FUNCTION_BLOCK alarmeHH_H_L_LL (* Composite Function Block Type *)
  (* Standard: 61499-2 *)
  (* Version 0.0, 1/23/2026, Schneider Electric, template *)
  PACKAGE Hidryco.HidrycoLib;
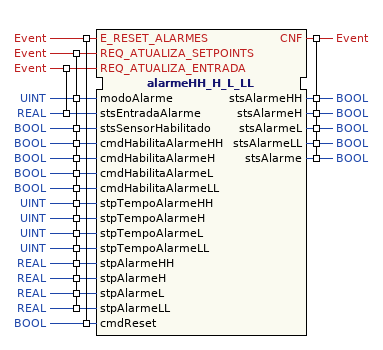
  EVENT_INPUT
    E_RESET_ALARMES WITH cmdReset;
    REQ_ATUALIZA_SETPOINTS WITH modoAlarme, cmdHabilitaAlarmeHH, cmdHabilitaAlarmeH, cmdHabilitaAlarmeL, cmdHabilitaAlarmeLL, stpTempoAlarmeHH, stpTempoAlarmeH, stpTempoAlarmeL, stpTempoAlarmeLL, stpAlarmeHH, stpAlarmeH, stpAlarmeL, stpAlarmeLL, stsSensorHabilitado;
    REQ_ATUALIZA_ENTRADA WITH stsEntradaAlarme;
  END_EVENT
  EVENT_OUTPUT
    CNF WITH stsAlarmeHH, stsAlarmeH, stsAlarmeL, stsAlarmeLL, stsAlarme; (* Execution Confirmation *)
  END_EVENT
  VAR_INPUT
    modoAlarme : UINT; (* 0 - AutoReset, 1 - Comando Reset *)
    stsEntradaAlarme : REAL;
    stsSensorHabilitado : BOOL;
    cmdHabilitaAlarmeHH : BOOL;
    cmdHabilitaAlarmeH : BOOL;
    cmdHabilitaAlarmeL : BOOL;
    cmdHabilitaAlarmeLL : BOOL;
    stpTempoAlarmeHH : UINT;
    stpTempoAlarmeH : UINT;
    stpTempoAlarmeL : UINT;
    stpTempoAlarmeLL : UINT;
    stpAlarmeHH : REAL;
    stpAlarmeH : REAL;
    stpAlarmeL : REAL;
    stpAlarmeLL : REAL;
    cmdReset : BOOL;
  END_VAR
  VAR_OUTPUT
    stsAlarmeHH : BOOL; (* Output event qualifier *)
    stsAlarmeH : BOOL;
    stsAlarmeL : BOOL;
    stsAlarmeLL : BOOL;
    stsAlarme : BOOL;
  END_VAR
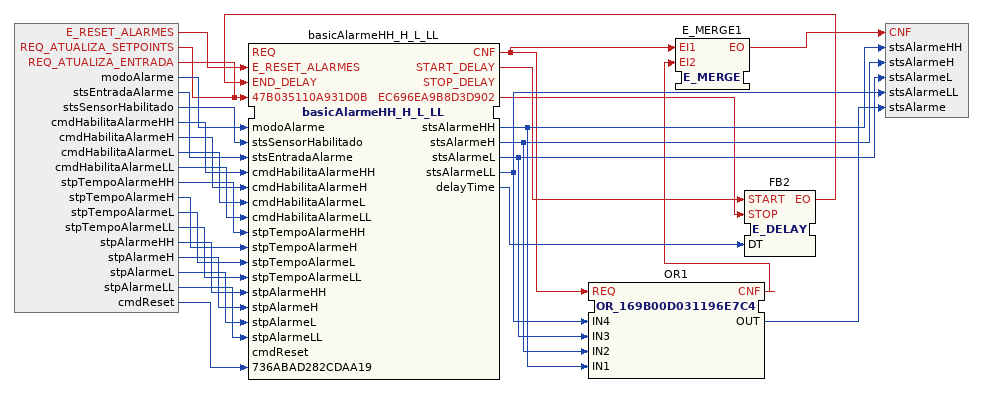
  FBS
    basicAlarmeHH_H_L_LL : basicAlarmeHH_H_L_LL;
    FB2 : E_DELAY;
    OR1 : OR_169B00D031196E7C4; {SET_ATTRIBUTE(Configuration.GenericFBType.InterfaceParams, Runtime.Standard#CNT:=4;OUT:BOOL)}
    E_MERGE1 : E_MERGE;
  END_FBS
  EVENT_CONNECTIONS
    basicAlarmeHH_H_L_LL.START_DELAY TO FB2.START;
    FB2.EO TO basicAlarmeHH_H_L_LL.END_DELAY;
    E_RESET_ALARMES TO basicAlarmeHH_H_L_LL.E_RESET_ALARMES;
    basicAlarmeHH_H_L_LL.CNF TO E_MERGE1.EI1;
    basicAlarmeHH_H_L_LL.CNF TO OR1.REQ;
    OR1.CNF TO E_MERGE1.EI2;
    E_MERGE1.EO TO CNF;
    REQ_ATUALIZA_SETPOINTS TO basicAlarmeHH_H_L_LL.47B035110A931D0B;
    REQ_ATUALIZA_ENTRADA TO basicAlarmeHH_H_L_LL.47B035110A931D0B;
    basicAlarmeHH_H_L_LL.EC696EA9B8D3D902 TO FB2.STOP;
  END_CONNECTIONS
  DATA_CONNECTIONS
    basicAlarmeHH_H_L_LL.delayTime TO FB2.DT;
    basicAlarmeHH_H_L_LL.stsAlarmeLL TO stsAlarmeLL;
    basicAlarmeHH_H_L_LL.stsAlarmeL TO stsAlarmeL;
    basicAlarmeHH_H_L_LL.stsAlarmeH TO stsAlarmeH;
    basicAlarmeHH_H_L_LL.stsAlarmeHH TO stsAlarmeHH;
    modoAlarme TO basicAlarmeHH_H_L_LL.modoAlarme;
    cmdHabilitaAlarmeHH TO basicAlarmeHH_H_L_LL.cmdHabilitaAlarmeHH;
    cmdHabilitaAlarmeH TO basicAlarmeHH_H_L_LL.cmdHabilitaAlarmeH;
    cmdHabilitaAlarmeL TO basicAlarmeHH_H_L_LL.cmdHabilitaAlarmeL;
    cmdHabilitaAlarmeLL TO basicAlarmeHH_H_L_LL.cmdHabilitaAlarmeLL;
    stpTempoAlarmeHH TO basicAlarmeHH_H_L_LL.stpTempoAlarmeHH;
    stpTempoAlarmeH TO basicAlarmeHH_H_L_LL.stpTempoAlarmeH;
    stpTempoAlarmeL TO basicAlarmeHH_H_L_LL.stpTempoAlarmeL;
    stpTempoAlarmeLL TO basicAlarmeHH_H_L_LL.stpTempoAlarmeLL;
    stpAlarmeHH TO basicAlarmeHH_H_L_LL.stpAlarmeHH;
    stpAlarmeH TO basicAlarmeHH_H_L_LL.stpAlarmeH;
    stpAlarmeL TO basicAlarmeHH_H_L_LL.stpAlarmeL;
    stpAlarmeLL TO basicAlarmeHH_H_L_LL.stpAlarmeLL;
    stsEntradaAlarme TO basicAlarmeHH_H_L_LL.stsEntradaAlarme;
    basicAlarmeHH_H_L_LL.stsAlarmeLL TO OR1.IN4;
    basicAlarmeHH_H_L_LL.stsAlarmeL TO OR1.IN3;
    basicAlarmeHH_H_L_LL.stsAlarmeH TO OR1.IN2;
    basicAlarmeHH_H_L_LL.stsAlarmeHH TO OR1.IN1;
    OR1.OUT TO stsAlarme;
    cmdReset TO basicAlarmeHH_H_L_LL.736ABAD282CDAA19;
    stsSensorHabilitado TO basicAlarmeHH_H_L_LL.stsSensorHabilitado;
  END_CONNECTIONS
END_FUNCTION_BLOCK
